Omron CX-Programmer project NuevoProyecto (CX-Programmer 9.54)

# PLC NuevoPLC1: CQM1 CPU41

## Program NuevoPrograma1 (no task)
Local symbols
EM 16.00 BOOL  ; EMERGENCIA
ET0 20.00 BOOL
ET1 20.01 BOOL
ET10 20.10 BOOL
ET11 20.11 BOOL
ET12 20.12 BOOL
ET13 20.13 BOOL
ET14 20.14 BOOL
ET15 20.15 BOOL
ET16 21.00 BOOL
ET17 21.01 BOOL
ET18 21.02 BOOL
ET19 21.03 BOOL
ET2 20.02 BOOL
ET20 21.04 BOOL
ET21 21.05 BOOL
ET22 21.06 BOOL
ET3 20.03 BOOL
ET4 20.04 BOOL
ET5 20.05 BOOL
ET6 20.06 BOOL
ET7 20.07 BOOL
ET8 20.08 BOOL
ET9 20.09 BOOL
FCB 0.04 BOOL
FCD 0.05 BOOL
FCE 0.07 BOOL
FCI 0.08 BOOL
FCN 0.06 BOOL
FCS 0.00 BOOL
LAVM1 100.15 BOOL  ; AVERIA M1
LAVM2 100.13 BOOL  ; AVERIA M2
LFM1 100.07 BOOL  ; LAMPARA FUNCIONAMIENTO M1
LFM2 100.01 BOOL  ; LAMPARA FUNCIONAMIENTO M2
M1DE 100.06 BOOL  ; M1 DERECHA
M1IZ 100.05 BOOL  ; M1 IZQUIERDA
M2B 100.08 BOOL  ; BAJAMOS M2
M2S 100.00 BOOL  ; SUBIMOS M2
PM 0.14 BOOL  ; PULSADOR MARCHA
PP 0.15 BOOL  ; PULSADOR PARO
PP_MOTORES 16.02 BOOL  ; PARAMOS LOS MOTORES
RESET_CONT 16.01 BOOL  ; RESET CONTADOR
RTM1 0.12 BOOL  ; RELE TERMICO M1
RTM2 0.13 BOOL  ; RELE TERMICO M2
SOB 100.11 BOOL  ; SOBRECARGA
S_T 0.11 BOOL  ; SENSOR DE TEMPERATURA

### Section PROG_PRINCIPAL

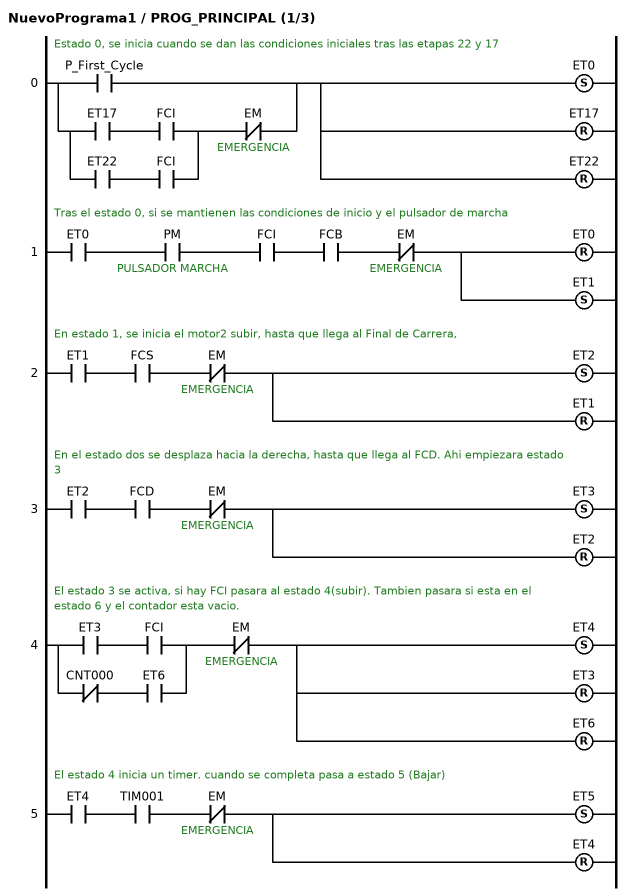
; rung 0: Estado 0, se inicia cuando se dan las condiciones iniciales tras las etapas 22 y 17
LD P_First_Cycle
LD ET17
AND FCI
LD ET22
AND FCI
ORLD
ANDNOT EM  ; EMERGENCIA
ORLD
SET ET0
RSET ET17
RSET ET22
; rung 1: Tras el estado 0, si se mantienen las condiciones de inicio y el pulsador de marcha
LD ET0
AND PM  ; PULSADOR MARCHA
AND FCI
AND FCB
ANDNOT EM  ; EMERGENCIA
RSET ET0
SET ET1
; rung 2: En estado 1, se inicia el motor2 subir, hasta que llega al Final de Carrera,
LD ET1
AND FCS
ANDNOT EM  ; EMERGENCIA
SET ET2
RSET ET1
; rung 3: En el estado dos se desplaza hacia la derecha, hasta que llega al FCD. Ahi empiezara estado 3
LD ET2
AND FCD
ANDNOT EM  ; EMERGENCIA
SET ET3
RSET ET2
; rung 4: El estado 3 se activa, si hay FCI pasara al estado 4(subir). Tambien pasara si esta en el estado 6 y el contador esta vacio.
LD ET3
AND FCI
LDNOT CNT000
AND ET6
ORLD
ANDNOT EM  ; EMERGENCIA
SET ET4
RSET ET3
RSET ET6
; rung 5: El estado 4 inicia un timer. cuando se completa pasa a estado 5 (Bajar)
LD ET4
AND TIM001
ANDNOT EM  ; EMERGENCIA
SET ET5
RSET ET4

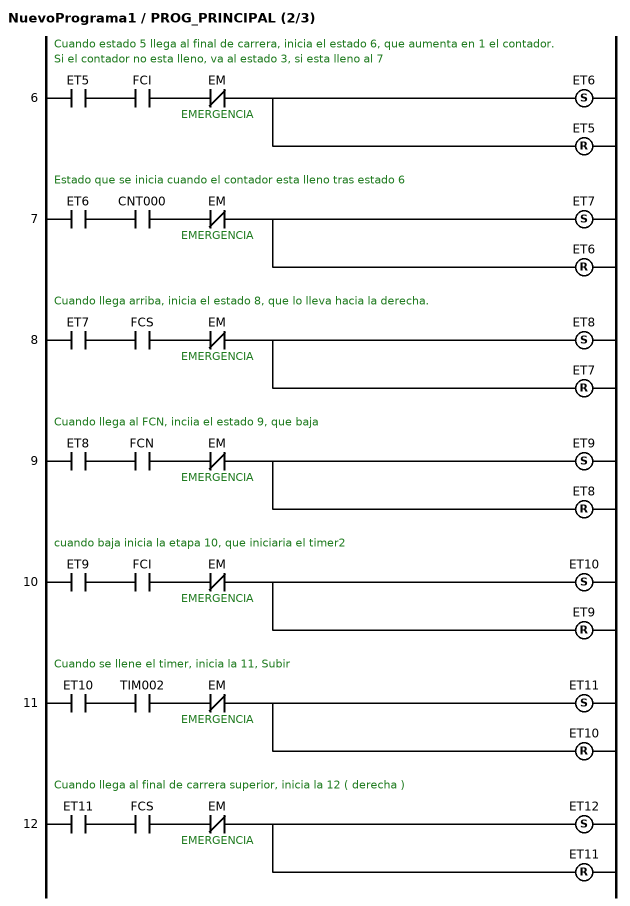
; rung 6: Cuando estado 5 llega al final de carrera, inicia el estado 6, que aumenta en 1 el contador. Si el contador no esta lleno, va al estado 3, si esta lleno al 7
LD ET5
AND FCI
ANDNOT EM  ; EMERGENCIA
SET ET6
RSET ET5
; rung 7: Estado que se inicia cuando el contador esta lleno tras estado 6
LD ET6
AND CNT000
ANDNOT EM  ; EMERGENCIA
SET ET7
RSET ET6
; rung 8: Cuando llega arriba, inicia el estado 8, que lo lleva hacia la derecha.
LD ET7
AND FCS
ANDNOT EM  ; EMERGENCIA
SET ET8
RSET ET7
; rung 9: Cuando llega al FCN, inciia el estado 9, que baja
LD ET8
AND FCN
ANDNOT EM  ; EMERGENCIA
SET ET9
RSET ET8
; rung 10: cuando baja inicia la etapa 10, que iniciaria el timer2
LD ET9
AND FCI
ANDNOT EM  ; EMERGENCIA
SET ET10
RSET ET9
; rung 11: Cuando se llene el timer, inicia la 11, Subir
LD ET10
AND TIM002
ANDNOT EM  ; EMERGENCIA
SET ET11
RSET ET10
; rung 12: Cuando llega al final de carrera superior, inicia la 12 ( derecha )
LD ET11
AND FCS
ANDNOT EM  ; EMERGENCIA
SET ET12
RSET ET11

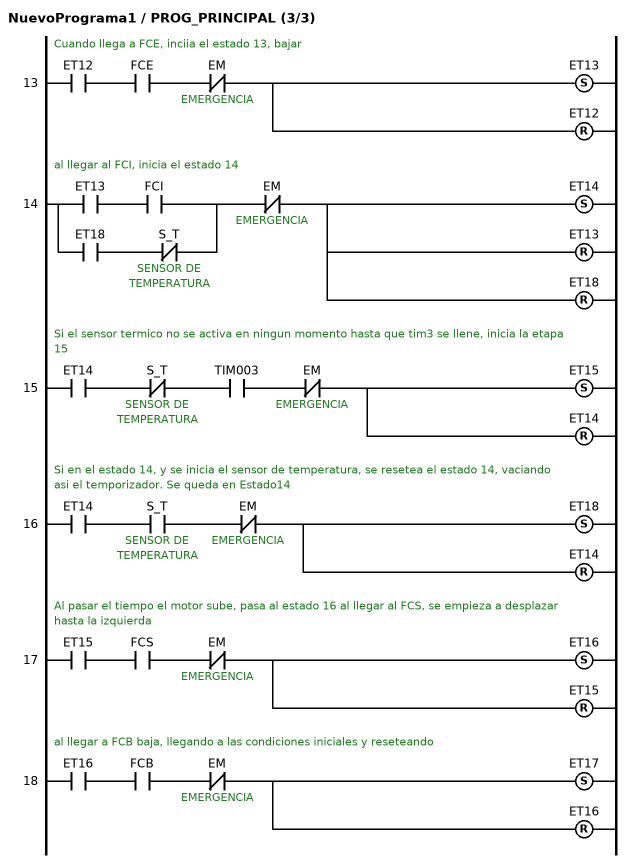
; rung 13: Cuando llega a FCE, inciia el estado 13, bajar
LD ET12
AND FCE
ANDNOT EM  ; EMERGENCIA
SET ET13
RSET ET12
; rung 14: al llegar al FCI, inicia el estado 14
LD ET13
AND FCI
LD ET18
ANDNOT S_T  ; SENSOR DE TEMPERATURA
ORLD
ANDNOT EM  ; EMERGENCIA
SET ET14
RSET ET13
RSET ET18
; rung 15: Si el sensor termico no se activa en ningun momento hasta que tim3 se llene, inicia la etapa 15
LD ET14
ANDNOT S_T  ; SENSOR DE TEMPERATURA
AND TIM003
ANDNOT EM  ; EMERGENCIA
SET ET15
RSET ET14
; rung 16: Si en el estado 14, y se inicia el sensor de temperatura, se resetea el estado 14, vaciando asi el temporizador. Se queda en Estado14
LD ET14
AND S_T  ; SENSOR DE TEMPERATURA
ANDNOT EM  ; EMERGENCIA
SET ET18
RSET ET14
; rung 17: Al pasar el tiempo el motor sube, pasa al estado 16 al llegar al FCS, se empieza a desplazar hasta la izquierda
LD ET15
AND FCS
ANDNOT EM  ; EMERGENCIA
SET ET16
RSET ET15
; rung 18: al llegar a FCB baja, llegando a las condiciones iniciales y reseteando
LD ET16
AND FCB
ANDNOT EM  ; EMERGENCIA
SET ET17
RSET ET16

### Section ETAPAS

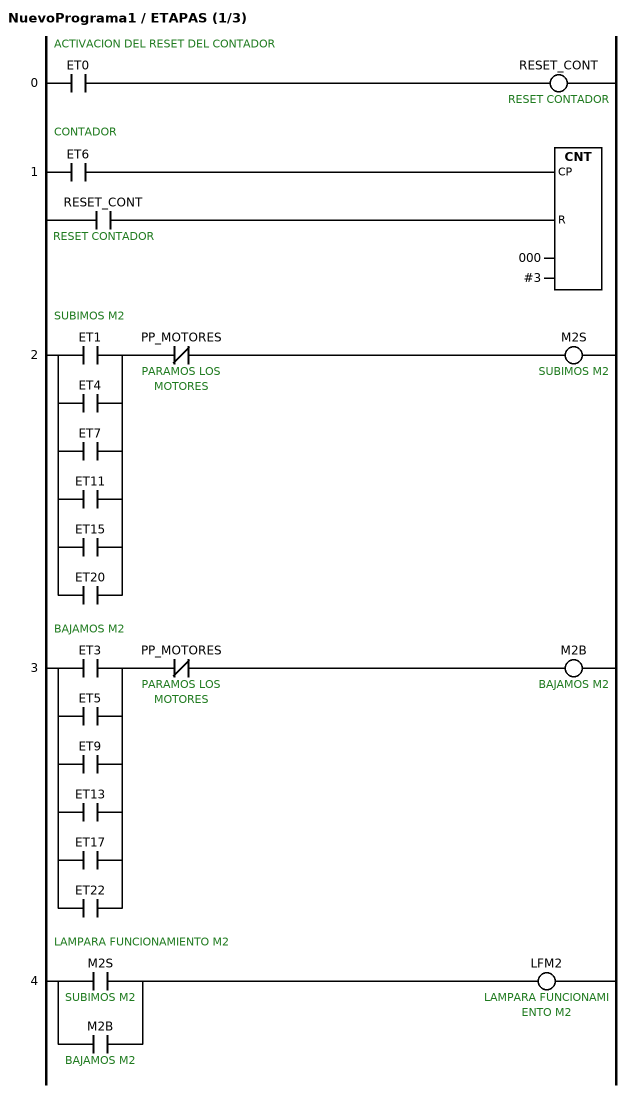
; rung 0: ACTIVACION DEL RESET DEL CONTADOR
LD ET0
OUT RESET_CONT  ; RESET CONTADOR
; rung 1: CONTADOR
LD ET6
LD RESET_CONT  ; RESET CONTADOR
CNT 000 #3
; rung 2: SUBIMOS M2
LD ET1
OR ET4
OR ET7
OR ET11
OR ET15
OR ET20
ANDNOT PP_MOTORES  ; PARAMOS LOS MOTORES
OUT M2S  ; SUBIMOS M2
; rung 3: BAJAMOS M2
LD ET3
OR ET5
OR ET9
OR ET13
OR ET17
OR ET22
ANDNOT PP_MOTORES  ; PARAMOS LOS MOTORES
OUT M2B  ; BAJAMOS M2
; rung 4: LAMPARA FUNCIONAMIENTO M2
LD M2S  ; SUBIMOS M2
OR M2B  ; BAJAMOS M2
OUT LFM2  ; LAMPARA FUNCIONAMIENTO M2

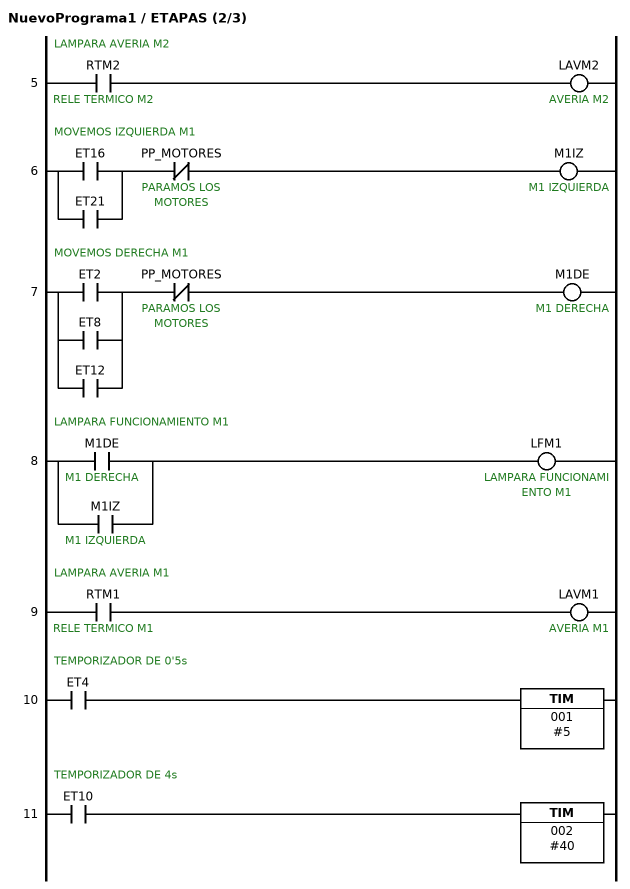
; rung 5: LAMPARA AVERIA M2
LD RTM2  ; RELE TERMICO M2
OUT LAVM2  ; AVERIA M2
; rung 6: MOVEMOS IZQUIERDA M1
LD ET16
OR ET21
ANDNOT PP_MOTORES  ; PARAMOS LOS MOTORES
OUT M1IZ  ; M1 IZQUIERDA
; rung 7: MOVEMOS DERECHA M1
LD ET2
OR ET8
OR ET12
ANDNOT PP_MOTORES  ; PARAMOS LOS MOTORES
OUT M1DE  ; M1 DERECHA
; rung 8: LAMPARA FUNCIONAMIENTO M1
LD M1DE  ; M1 DERECHA
OR M1IZ  ; M1 IZQUIERDA
OUT LFM1  ; LAMPARA FUNCIONAMIENTO M1
; rung 9: LAMPARA AVERIA M1
LD RTM1  ; RELE TERMICO M1
OUT LAVM1  ; AVERIA M1
; rung 10: TEMPORIZADOR DE 0'5s
LD ET4
TIM 001 #5
; rung 11: TEMPORIZADOR DE 4s
LD ET10
TIM 002 #40

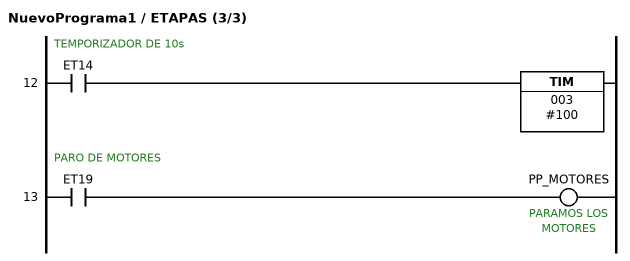
; rung 12: TEMPORIZADOR DE 10s
LD ET14
TIM 003 #100
; rung 13: PARO DE MOTORES
LD ET19
OUT PP_MOTORES  ; PARAMOS LOS MOTORES

### Section EMERGENCIA

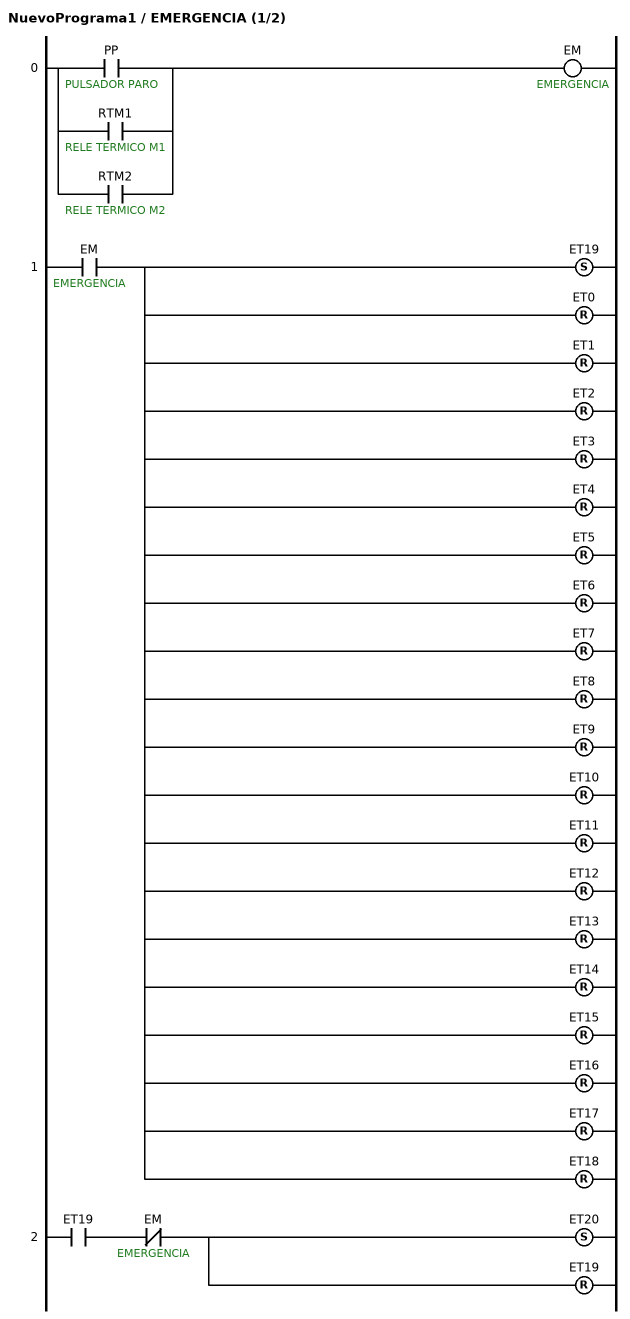
; rung 0
LD PP  ; PULSADOR PARO
OR RTM1  ; RELE TERMICO M1
OR RTM2  ; RELE TERMICO M2
OUT EM  ; EMERGENCIA
; rung 1
LD EM  ; EMERGENCIA
SET ET19
RSET ET0
RSET ET1
RSET ET2
RSET ET3
RSET ET4
RSET ET5
RSET ET6
RSET ET7
RSET ET8
RSET ET9
RSET ET10
RSET ET11
RSET ET12
RSET ET13
RSET ET14
RSET ET15
RSET ET16
RSET ET17
RSET ET18
; rung 2
LD ET19
ANDNOT EM  ; EMERGENCIA
SET ET20
RSET ET19

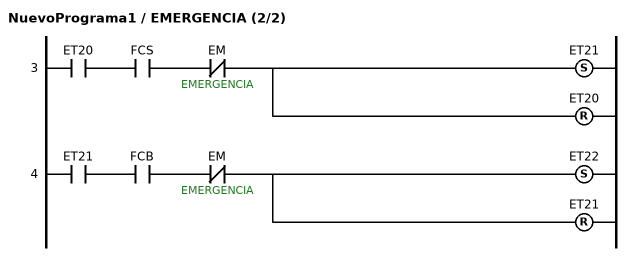
; rung 3
LD ET20
AND FCS
ANDNOT EM  ; EMERGENCIA
SET ET21
RSET ET20
; rung 4
LD ET21
AND FCB
ANDNOT EM  ; EMERGENCIA
SET ET22
RSET ET21

### Section END
; rung 0
END(01)